(* IEC 61131-3 sources: Industry-PLC-LLM/data/PLCBEAD_repo/PLCBEAD_PLCEmbed-main/PLC-BEAD/Source/GEB/BIT_TOGGLE_B, 1 file *)

(* ---- BIT_TOGGLE_B.ST ---- *)
FUNCTION BIT_TOGGLE_B:BYTE
	VAR_INPUT
		IN :	BYTE;
		POS :	INT;
	END_VAR

	BIT_TOGGLE_B := SHL(BYTE#1, POS) XOR IN;
END_FUNCTION

PROGRAM program0
  VAR
    LocalVar0 : BYTE;
    LocalVaR1  : INT;
    CEIL5_OUT : BYTE;
  END_VAR

  CEIL5_OUT := BIT_TOGGLE_B(LocalVar0, LocalVaR1 );
END_PROGRAM
